FUNCTION_BLOCK FB_Obj_AddParam EXTENDS FB_BA_View
VAR
	TestSpVal			: FB_UDef_SpVal				:= (iParent:=THIS^,		sDescription:='My user defined setpoint object',				eMode:=E_UDef_Mode.eAdd);
	TestSpValEx			: FB_UDef_SpValEx			:= (iParent:=THIS^,		sDescription:='Another user defined enabled setpoint object',	eMode:=E_UDef_Mode.eSubstract);
	
	TestBValEx			: FB_UDef_BValEx			:= (iParent:=THIS^,		sDescription:='My user defined boolean value extension');
END_VAR
VAR
	{region 'Test'}
		nOffset			: UINT						:= 3;
	{endregion}
END_VAR

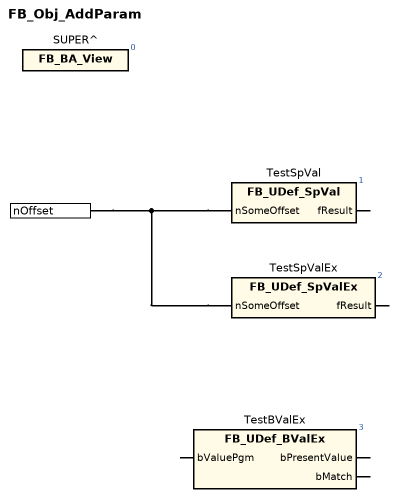
SUPER^(); // FB_BA_View
TestSpVal(nSomeOffset := nOffset); // FB_UDef_SpVal
TestSpValEx(nSomeOffset := nOffset); // FB_UDef_SpValEx
TestBValEx(); // FB_UDef_BValEx

END_FUNCTION_BLOCK

(* stored: Version 1.1.0.1, ProductVersion 3.1.4024.11
   POU FB_Obj_AddParam: Id {ee9c847e-86ab-4ab1-a8c8-e6dfc4e4d446}, SpecialFunc None *)
